//{{V2}}
ORGANIZATION_BLOCK OB1
TITLE= "Cyclic main program"


AUTHOR:nb
FAMILY:nb
NAME:nb
VERSION:1.0


VAR_TEMP
       OB1_EV_CLASS:BYTE //Bits 0-3 = 1 (Coming event), Bits 4-7 = 1 (Event class 1)
       OB1_SCAN_1:BYTE //1 (Cold restart scan 1 of OB 1), 3 (Scan 2-n of OB 1)
       OB1_PRIORITY:BYTE //1 (Priority of 1 is lowest)
       OB1_OB_NUMBR:BYTE //1 (Organization block 1, OB1)
       OB1_RESERVED_1:BYTE //Reserved for system
       OB1_RESERVED_2:BYTE //Reserved for system
       OB1_PREV_CYCLE:INT //Cycle time of previous OB1 scan (milliseconds)
       OB1_MIN_CYCLE:INT //Minimum cycle time of OB1 (milliseconds)
       OB1_MAX_CYCLE:INT //Maximum cycle time of OB1 (milliseconds)
       OB1_DATE_TIME:DATE_AND_TIME //Date and time OB1 started
END_VAR
BEGIN

NETWORK
TITLE=Linja e Start,Stop,Run,Emergjenca dhe dritat e Start && Reset
//{{k}}
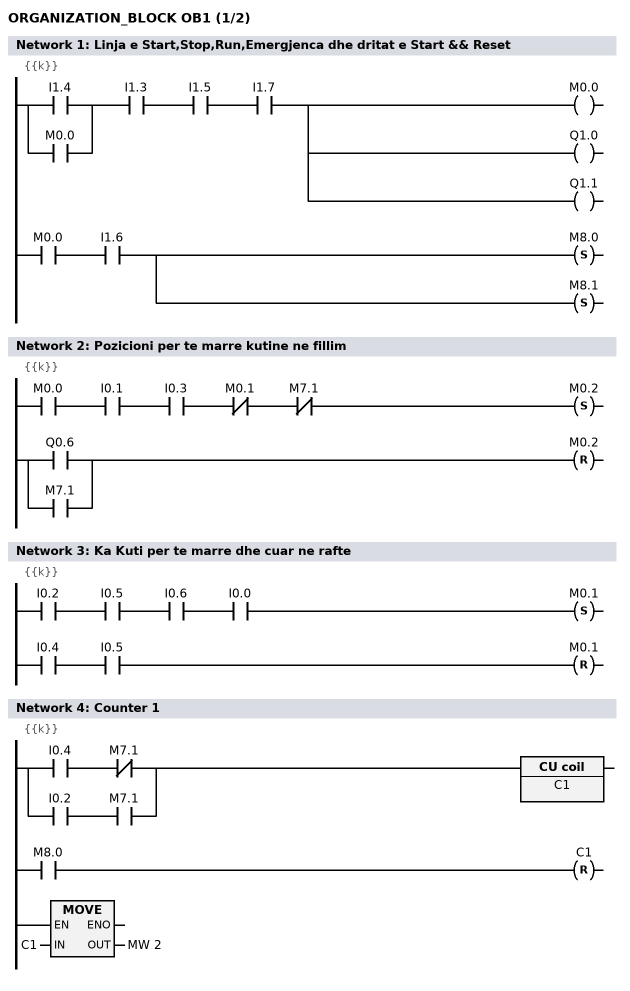

       A(
       O    I1.4
       O    M0.0
       )
       A    I1.3
       A    I1.5
       A    I1.7
       =    M0.0
       =    Q1.0
       =    Q1.1
       A    M0.0
       A    I1.6
       S    M8.0
       S    M8.1
NETWORK
TITLE=Pozicioni per te marre kutine ne fillim
//{{k}}

       A    M0.0
       A    I0.1
       A    I0.3
       AN   M0.1
       AN   M7.1
       S    M0.2
       A(
       O    Q0.6
       O    M7.1
       )
       R    M0.2
NETWORK
TITLE=Ka Kuti per te marre dhe cuar ne rafte
//{{k}}

       A    I0.2
       A    I0.5
       A    I0.6
       A    I0.0
       S    M0.1
       A    I0.4
       A    I0.5
       R    M0.1
NETWORK
TITLE=Counter 1
//{{k}}

       A    I0.4
       AN   M7.1
       O
       A    I0.2
       A    M7.1
       CU   C1
       BLD  101
       NOP  0
       NOP  0
       A    M8.0
       R    C1
       L    C1
       T    MW        2
       NOP  0
       NOP  0
NETWORK
TITLE=Timer per A6 dhe A7
//{{k}}
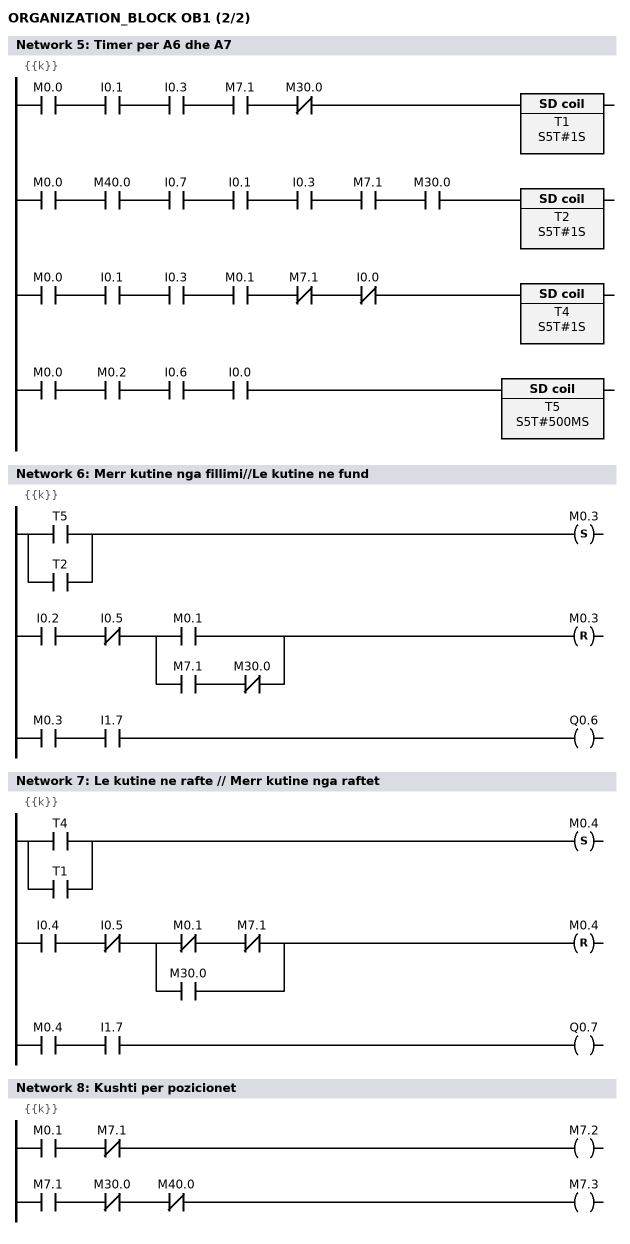

       A    M0.0
       A    I0.1
       A    I0.3
       A    M7.1
       AN   M30.0
       L    S5T#1S
       SD   T1
       A    M0.0
       A    M40.0
       A    I0.7
       A    I0.1
       A    I0.3
       A    M7.1
       A    M30.0
       L    S5T#1S
       SD   T2
       A    M0.0
       A    I0.1
       A    I0.3
       A    M0.1
       AN   M7.1
       AN   I0.0
       L    S5T#1S
       SD   T4
       A    M0.0
       A    M0.2
       A    I0.6
       A    I0.0
       L    S5T#500MS
       SD   T5
NETWORK
TITLE=Merr kutine nga fillimi//Le kutine ne fund
//{{k}}

       O    T5
       O    T2
       S    M0.3
       A    I0.2
       AN   I0.5
       A(
       A    M0.1
       O
       A    M7.1
       AN   M30.0
       )
       R    M0.3
       A    M0.3
       A    I1.7
       =    Q0.6
NETWORK
TITLE=Le kutine ne rafte // Merr kutine nga raftet
//{{k}}

       O    T4
       O    T1
       S    M0.4
       A    I0.4
       AN   I0.5
       A(
       AN   M0.1
       AN   M7.1
       O    M30.0
       )
       R    M0.4
       A    M0.4
       A    I1.7
       =    Q0.7
NETWORK
TITLE=Kushti per pozicionet
//{{k}}

       A    M0.1
       AN   M7.1
       =    M7.2
       A    M7.1
       AN   M30.0
       AN   M40.0
       =    M7.3
NETWORK
TITLE=Pozicioni 1
//{{k}}

       A(
       A    M0.0
       A(
       L    MW        2
       L    0
       ==I
       )
       A    I0.3
       A(
       O    M7.2
       O    M7.3
       )
       S    M0.5
       A    M0.0
       A(
       O    M0.2
       O    M30.0
       )
       )
       R    M0.5
       NOP  0
NETWORK
TITLE=Pozicioni 2
//{{k}}

       A(
       A    M0.0
       A(
       L    MW        2
       L    1
       ==I
       )
       A    I0.3
       A(
       O    M7.2
       O    M7.3
       )
              S    M0.6
       A    M0.0
       A(
       O    M0.2
       O    M30.0
       )
       )
       R    M0.6
       NOP  0
NETWORK
TITLE=Pozicioni 3
//{{k}}

       A(
       A(
       A    M0.0
       A(
       L    MW        2
       L    2
       ==I
       )
       A    I0.3
       A(
       O    M7.2
       O    M7.3
       )

       )
       S    M0.7
       A    M0.0
       A(
       O    M0.2
       O    M30.0
       )
       )
       R    M0.7
       NOP  0
NETWORK
TITLE=Pozicioni 4
//{{k}}

       A(
       A(
       A    M0.0
       A(
       L    MW        2
       L    3
       ==I
       )
       A    I0.3
       A(
       O    M7.2
       O    M7.3
       )
       )
       S    M1.0
       A    M0.0
       A(
       O    M0.2
       O    M30.0
       )
       )
       R    M1.0
       NOP  0
NETWORK
TITLE=Pozicioni 5
//{{k}}

       A(
       A(
       A    M0.0
       A(
       L    MW        2
       L    4
       ==I
       )
       A    I0.3
       A(
       O    M7.2
       O    M7.3
       )

       )
       S    M1.1
       A    M0.0
       A(
       O    M0.2
       O    M30.0
       )
       )
       R    M1.1
       NOP  0
NETWORK
TITLE=Pozicioni 6
//{{k}}

       A(
       A(
       A    M0.0
       A(
       L    MW        2
       L    5
       ==I
       )
       A    I0.3
       A(
       O    M7.2
       O    M7.3
       )

             )
       S    M1.2
       A    M0.0
       A(
       O    M0.2
       O    M30.0
       )
       )
       R    M1.2
       NOP  0
NETWORK
TITLE=Pozicioni 7
//{{k}}

       A(
       A(
       A    M0.0
       A(
       L    MW        2
       L    6
       ==I
       )
       A    I0.3
       A(
       O    M7.2
       O    M7.3
       )


       )
       S    M1.3
       A    M0.0
       A(
       O    M0.2
       O    M30.0
       )
       )
       R    M1.3
       NOP  0
NETWORK
TITLE=Pozicioni 8
//{{k}}

       A(
       A(
       A    M0.0
       A(
       L    MW        2
       L    7
       ==I
       )
       A    I0.3
       A(
       O    M7.2
       O    M7.3
       )


       )
       S    M1.4
       A    M0.0
       A(
       O    M0.2
       O    M30.0
       )
       )
       R    M1.4
       NOP  0
NETWORK
TITLE=Pozicioni 9
//{{k}}

       A(
       A(
       A    M0.0
       A(
       L    MW        2
       L    8
       ==I
       )
       A    I0.3
       A(
       O    M7.2
       O    M7.3
       )


       )
       S    M1.5
       A    M0.0
       A(
       O    M0.2
       O    M30.0
       )
       )
       R    M1.5
       NOP  0
NETWORK
TITLE=Pozicioni 10
//{{k}}

       A(
       A(
       A    M0.0
       A(
       L    MW        2
       L    9
       ==I
       )
       A    I0.3
       A(
       O    M7.2
       O    M7.3
       )

       )
       S    M1.6
       A    M0.0
       A(
       O    M0.2
       O    M30.0
       )
       )
       R    M1.6
       NOP  0
NETWORK
TITLE=Pozicioni 11
//{{k}}

       A(
       A(
       A    M0.0
       A(
       L    MW        2
       L    10
       ==I
       )
       A    I0.3
       A(
       O    M7.2
       O    M7.3
       )


       )
       S    M1.7
       A    M0.0
       A(
       O    M0.2
       O    M30.0
       )
       )
       R    M1.7
       NOP  0
NETWORK
TITLE=Pozicioni 12
//{{k}}

       A(
       A(
       A    M0.0
       A(
       L    MW        2
       L    11
       ==I
       )
       A    I0.3
       A(
       O    M7.2
       O    M7.3
       )

              )
       S    M2.0
       A    M0.0
       A(
       O    M0.2
       O    M30.0
       )
       )
       R    M2.0
       NOP  0
NETWORK
TITLE=Pozicioni 13
//{{k}}

       A(
       A(
       A    M0.0
       A(
       L    MW        2
       L    12
       ==I
       )
       A    I0.3
       A(
       O    M7.2
       O    M7.3
       )


       )
       S    M2.1
       A    M0.0
       A(
       O    M0.2
       O    M30.0
       )
       )
       R    M2.1
       NOP  0
NETWORK
TITLE=Pozicioni 14
//{{k}}

       A(
       A(
       A    M0.0
       A(
       L    MW        2
       L    13
       ==I
       )
       A    I0.3
       A(
       O    M7.2
       O    M7.3
       )

       )
       S    M2.2
       A    M0.0
       A(
       O    M0.2
       O    M30.0
       )
       )
       R    M2.2
       NOP  0
NETWORK
TITLE=Pozicioni 15
//{{k}}

       A(
       A(
       A    M0.0
       A(
       L    MW        2
       L    14
       ==I
       )
       A    I0.3
       A(
       O    M7.2
       O    M7.3
       )

       )
       S    M2.3
       A    M0.0
       A(
       O    M0.2
       O    M30.0
       )
       )
       R    M2.3
       NOP  0
NETWORK
TITLE=Pozicioni 16
//{{k}}

       A(
       A(
       A    M0.0
       A(
       L    MW        2
       L    15
       ==I
       )
       A    I0.3
       A(
       O    M7.2
       O    M7.3
       )


       )
       S    M2.4
       A    M0.0
       A(
       O    M0.2
       O    M30.0
       )
       )
       R    M2.4
       NOP  0
NETWORK
TITLE=Pozicioni 17
//{{k}}

       A(
       A(
       A    M0.0
       A(
       L    MW        2
       L    16
       ==I
       )
       A    I0.3
       A(
       O    M7.2
       O    M7.3
       )


       )
       S    M2.5
       A    M0.0
       A(
       O    M0.2
       O    M30.0
       )
       )
       R    M2.5
       NOP  0
NETWORK
TITLE=Pozicioni 18
//{{k}}

       A(
       A(
       A    M0.0
       A(
       L    MW        2
       L    17
       ==I
       )
       A    I0.3
       A(
       O    M7.2
       O    M7.3
       )


       )
       S    M2.6
       A    M0.0
       A(
       O    M0.2
       O    M30.0
       )
       )
       R    M2.6
       NOP  0
NETWORK
TITLE=Pozicioni 19
//{{k}}

       A(
       A(
       A    M0.0
       A(
       L    MW        2
       L    18
       ==I
       )
       A    I0.3
       A(
       O    M7.2
       O    M7.3
       )


       )
       S    M2.7
       A    M0.0
       A(
       O    M0.2
       O    M30.0
       )
       )
       R    M2.7
       NOP  0
NETWORK
TITLE=Pozicioni 20
//{{k}}

       A(
       A(
       A    M0.0
       A(
       L    MW        2
       L    19
       ==I
       )
       A    I0.3
       A(
       O    M7.2
       O    M7.3
       )


       )
       S    M10.0
       A    M0.0
       A(
       O    M0.2
       O    M30.0
       )
       )
       R    M10.0
       NOP  0
NETWORK
TITLE=Pozicioni 21
//{{k}}

       A(
       A(
       A    M0.0
       A(
       L    MW        2
       L    20
       ==I
       )
       A    I0.3
       A(
       O    M7.2
       O    M7.3
       )

             )
       S    M10.1
       A    M0.0
       A(
       O    M0.2
       O    M30.0
       )
       )
       R    M10.1
       NOP  0
NETWORK
TITLE=Pozicioni 22
//{{k}}

       A(
       A(
       A    M0.0
       A(
       L    MW        2
       L    21
       ==I
       )
       A    I0.3
       A(
       O    M7.2
       O    M7.3
       )


       )
       S    M10.2
       A    M0.0
       A(
       O    M0.2
       O    M30.0
       )
       )
       R    M10.2
       NOP  0
NETWORK
TITLE=Pozicioni 23
//{{k}}

       A(
       A(
       A    M0.0
       A(
       L    MW        2
       L    22
       ==I
       )
       A    I0.3
       A(
       O    M7.2
       O    M7.3
       )


       )
       S    M10.3
       A    M0.0
       A(
       O    M0.2
       O    M30.0
       )
       )
       R    M10.3
       NOP  0
NETWORK
TITLE=Pozicioni 24
//{{k}}

       A(
       A(
       A    M0.0
       A(
       L    MW        2
       L    23
       ==I
       )
       A    I0.3
       A(
       O    M7.2
       O    M7.3
       )


       )
       S    M10.4
       A    M0.0
       A(
       O    M0.2
       O    M30.0
       )
       )
       R    M10.4
       NOP  0
NETWORK
TITLE=Pozicioni 25
//{{k}}

       A(
       A(
       A    M0.0
       A(
       L    MW        2
       L    24
       ==I
       )
       A    I0.3
       A(
       O    M7.2
       O    M7.3
       )


       )
       S    M10.5
       A    M0.0
       A(
       O    M0.2
       O    M30.0
       )
       )
       R    M10.5
       NOP  0
NETWORK
TITLE=Pozicioni 26
//{{k}}

       A(
       A(
       A    M0.0
       A(
       L    MW        2
       L    25
       ==I
       )
       A    I0.3
       A(
       O    M7.2
       O    M7.3
       )


       )
       S    M10.6
       A    M0.0
       A(
       O    M0.2
       O    M30.0
       )
       )
       R    M10.6
       NOP  0
NETWORK
TITLE=Pozicioni 27
//{{k}}

       A(
       A(
       A    M0.0
       A(
       L    MW        2
       L    26
       ==I
       )
       A    I0.3
       A(
       O    M7.2
       O    M7.3
       )

              )
       S    M10.7
       A    M0.0
       A(
       O    M0.2
       O    M30.0
       )
       )
       R    M10.7
       NOP  0
NETWORK
TITLE=Pozicioni 28
//{{k}}

       A(
       A(
       A    M0.0
       A(
       L    MW        2
       L    27
       ==I
       )
       A    I0.3
       A(
       O    M7.2
       O    M7.3
       )


       )
       S    M4.0
       A    M0.0
       A(
       O    M0.2
       O    M30.0
       )
       )
       R    M4.0
       NOP  0
NETWORK
TITLE=Pozicioni 29
//{{k}}

       A(
       A(
       A    M0.0
       A(
       L    MW        2
       L    28
       ==I
       )
       A    I0.3
       A(
       O    M7.2
       O    M7.3
       )


       )
       S    M4.1
       A    M0.0
       A(
       O    M0.2
       O    M30.0
       )
       )
       R    M4.1
       NOP  0
NETWORK
TITLE=Pozicioni 30
//{{k}}

       A(
       A(
       A    M0.0
       A(
       L    MW        2
       L    29
       ==I
       )
       A    I0.3
       A(
       O    M7.2
       O    M7.3
       )


       )
       S    M4.2
       A    M0.0
       A(
       O    M0.2
       O    M30.0
       )
       )
       R    M4.2
       NOP  0
NETWORK
TITLE=Pozicioni 31
//{{k}}

       A(
       A(
       A    M0.0
       A(
       L    MW        2
       L    30
       ==I
       )
       A    I0.3
       A(
       O    M7.2
       O    M7.3
       )

       )
       S    M4.3
       A    M0.0
       A(
       O    M0.2
       O    M30.0
       )
       )
       R    M4.3
       NOP  0
NETWORK
TITLE=Pozicioni 32
//{{k}}

       A(
       A(
       A    M0.0
       A(
       L    MW        2
       L    31
       ==I
       )
       A    I0.3
       A(
       O    M7.2
       O    M7.3
       )

       )
       S    M4.4
       A    M0.0
       A(
       O    M0.2
       O    M30.0
       )
       )
       R    M4.4
       NOP  0
NETWORK
TITLE=Pozicioni 33
//{{k}}

       A(
       A(
       A    M0.0
       A(
       L    MW        2
       L    32
       ==I
       )
       A    I0.3
       A(
       O    M7.2
       O    M7.3
       )

       )
       S    M4.5
       A    M0.0
       A(
       O    M0.2
       O    M30.0
       )
       )
       R    M4.5
       NOP  0
NETWORK
TITLE=Pozicioni 34
//{{k}}

       A(
       A(
       A    M0.0
       A(
       L    MW        2
       L    33
       ==I
       )
       A    I0.3
       A(
       O    M7.2
       O    M7.3
       )

       )
       S    M4.6
       A    M0.0
       A(
       O    M0.2
       O    M30.0
       )
       )
       R    M4.6
       NOP  0
NETWORK
TITLE=Pozicioni 35
//{{k}}

       A(
       A(
       A    M0.0
       A(
       L    MW        2
       L    34
       ==I
       )
       A    I0.3
       A(
       O    M7.2
       O    M7.3
       )

       )
       S    M4.7
       A    M0.0
       A(
       O    M0.2
       O    M30.0
       )
       )
       R    M4.7
       NOP  0
NETWORK
TITLE=Pozicioni 36
//{{k}}

       A(
       A(
       A    M0.0
       A(
       L    MW        2
       L    35
       ==I
       )
       A    I0.3
       A(
       O    M7.2
       O    M7.3
       )


       )
       S    M5.0
       A    M0.0
       A(
       O    M0.2
       O    M30.0
       )
       )
       R    M5.0
       NOP  0
NETWORK
TITLE=Pozicioni 37
//{{k}}

       A(
       A(
       A    M0.0
       A(
       L    MW        2
       L    36
       ==I
       )
       A    I0.3
       A(
       O    M7.2
       O    M7.3
       )


       )
       S    M5.1
       A    M0.0
       A(
       O    M0.2
       O    M30.0
       )
       )
       R    M5.1
       NOP  0
NETWORK
TITLE=Pozicioni 38
//{{k}}

       A(
       A(
       A    M0.0
       A(
       L    MW        2
       L    37
       ==I
       )
       A    I0.3
       A(
       O    M7.2
       O    M7.3
       )


       )
       S    M5.2
       A    M0.0
       A(
       O    M0.2
       O    M30.0
       )
       )
       R    M5.2
       NOP  0
NETWORK
TITLE=Pozicioni 39
//{{k}}

       A(
       A(
       A    M0.0
       A(
       L    MW        2
       L    38
       ==I
       )

       A    I0.3
       A(
       O    M7.2
       O    M7.3
       )

       )

       S    M5.3
       A    M0.0
       A(
       O    M0.2
       O    M30.0
       )
       )
       R    M5.3
       NOP  0
NETWORK
TITLE=Pozicioni 40
//{{k}}

       A(
       A(
       A    M0.0
       A(
       L    MW        2
       L    39
       ==I
       )
       A    I0.3
       A(
       O    M7.2
       O    M7.3
       )

             )
       S    M5.4
       A    M0.0
       A(
       O    M0.2
       O    M30.0
       )
       )
       R    M5.4
       NOP  0
NETWORK
TITLE=Pozicioni 41
//{{k}}

       A(
       A(
       A    M0.0
       A(
       L    MW        2
       L    40
       ==I
       )
       A    I0.3
       A(
       O    M7.2
       O    M7.3
       )

       )
       S    M5.5
       A    M0.0
       A(
       O    M0.2
       O    M30.0
       )
       )
       R    M5.5
       NOP  0
NETWORK
TITLE=Pozicioni 42
//{{k}}

       A(
       A(
       A    M0.0
       A(
       L    MW        2
       L    41
       ==I
       )
       A    I0.3
       A(
       O    M7.2
       O    M7.3
       )

             )
       S    M5.6
       A    M0.0
       A(
       O    M0.2
       O    M30.0
       )
       )
       R    M5.6
       NOP  0
NETWORK
TITLE=Pozicioni 43
//{{k}}

       A(
       A(
       A    M0.0
       A(
       L    MW        2
       L    42
       ==I
       )
       A    I0.3
       A(
       O    M7.2
       O    M7.3
       )

              )
       S    M5.7
       A    M0.0
       A(
       O    M0.2
       O    M30.0
       )
       )
       R    M5.7
       NOP  0
NETWORK
TITLE=Pozicioni 44
//{{k}}

       A(
       A(
       A    M0.0
       A(
       L    MW        2
       L    43
       ==I
       )
       A    I0.3
       A(
       O    M7.2
       O    M7.3
       )

              )
       S    M6.0
       A    M0.0
       A(
       O    M0.2
       O    M30.0
       )
       )
       R    M6.0
       NOP  0
NETWORK
TITLE=Pozicioni 45
//{{k}}

       A(
       A(
       A    M0.0
       A(
       L    MW        2
       L    44
       ==I
       )
       A    I0.3
       A(
       O    M7.2
       O    M7.3
       )


       )
       S    M6.1
       A    M0.0
       A(
       O    M0.2
       O    M30.0
       )
       )
       R    M6.1
       NOP  0
NETWORK
TITLE=Pozicioni 46
//{{k}}

       A(
       A(
       A    M0.0
       A(
       L    MW        2
       L    45
       ==I
       )
       A    I0.3
       A(
       O    M7.2
       O    M7.3
       )

              )
       S    M6.2
       A    M0.0
       A(
       O    M0.2
       O    M30.0
       )
       )
       R    M6.2
       NOP  0
NETWORK
TITLE=Pozicioni 47
//{{k}}

       A(
       A(
       A    M0.0
       A(
       L    MW        2
       L    46
       ==I
       )
       A    I0.3
       A(
       O    M7.2
       O    M7.3
       )

              )
       S    M6.3
       A    M0.0
       A(
       O    M0.2
       O    M30.0
       )
       )
       R    M6.3
       NOP  0
NETWORK
TITLE=Pozicioni 48
//{{k}}

       A(
       A(
       A    M0.0
       A(
       L    MW        2
       L    47
       ==I
       )
       A    I0.3
       A(
       O    M7.2
       O    M7.3
       )


       )
       S    M6.4
       A    M0.0
       A(
       O    M0.2
       O    M30.0
       )
       )
       R    M6.4
       NOP  0
NETWORK
TITLE=Pozicioni 49
//{{k}}

       A(
       A(
       A    M0.0
       A(
       L    MW        2
       L    48
       ==I
       )
       A    I0.3
       A(
       O    M7.2
       O    M7.3
       )


       )
       S    M6.5
       A    M0.0
       A(
       O    M0.2
       O    M30.0
       )
       )
       R    M6.5
       NOP  0
NETWORK
TITLE=Pozicioni 50
//{{k}}

       A(
       A(
       A    M0.0
       A(
       L    MW        2
       L    49
       ==I
       )
       A    I0.3
       A(
       O    M7.2
       O    M7.3
       )

             )
       S    M6.6
       A    M0.0
       A(
       O    M0.2
       O    M30.0
       )
       )
       R    M6.6
       NOP  0
NETWORK
TITLE=Actuator 0
//{{k}}
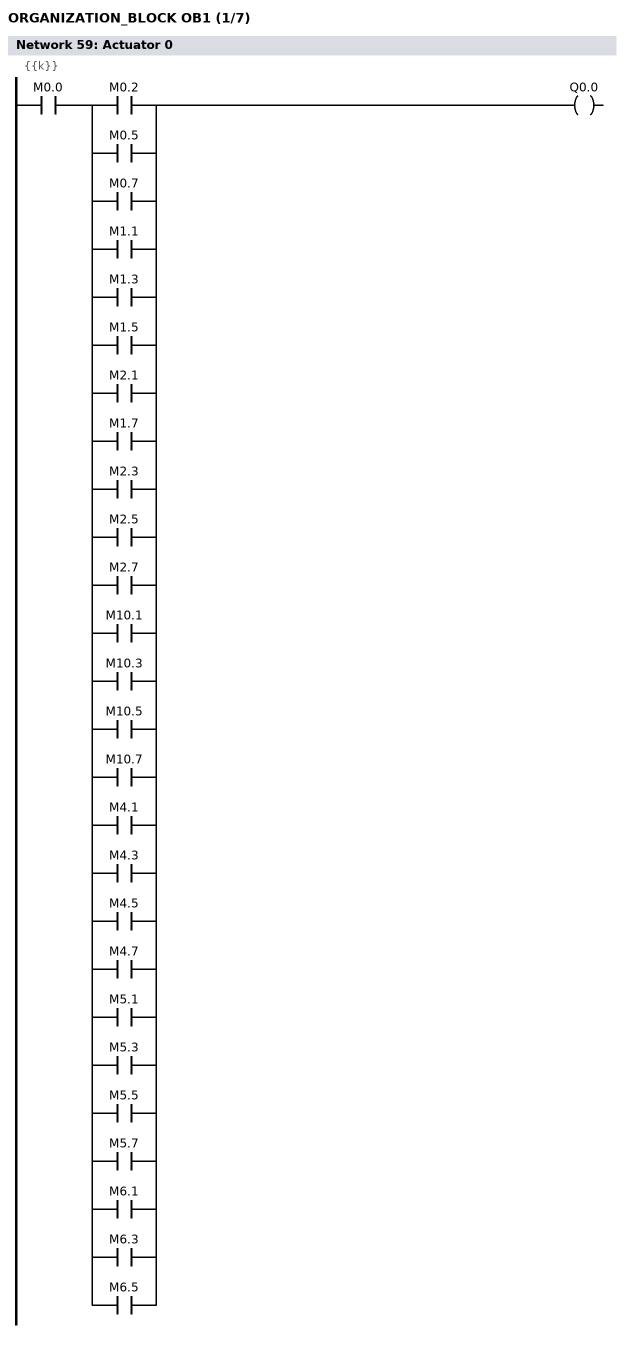

       A    M0.0
       A(
       O    M0.2
       O    M0.5
       O    M0.7
       O    M1.1
       O    M1.3
       O    M1.5
       O    M2.1
       O    M1.7
       O    M2.3
       O    M2.5
       O    M2.7
       O    M10.1
       O    M10.3
       O    M10.5
       O    M10.7
       O    M4.1
       O    M4.3
       O    M4.5
       O    M4.7
       O    M5.1
       O    M5.3
       O    M5.5
       O    M5.7
       O    M6.1
       O    M6.3
       O    M6.5
       )
       =    Q0.0
NETWORK
TITLE=Actuator 1
//{{k}}
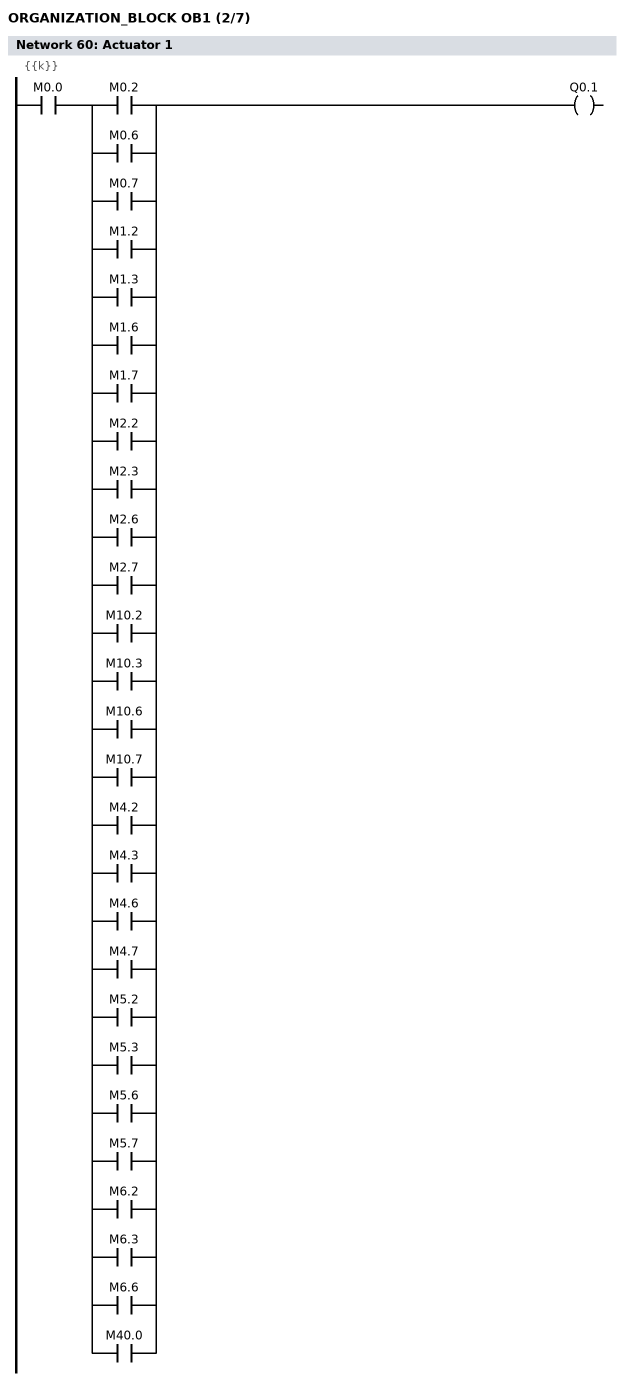

       A    M0.0
       A(
       O    M0.2
       O    M0.6
       O    M0.7
       O    M1.2
       O    M1.3
       O    M1.6
       O    M1.7
       O    M2.2
       O    M2.3
       O    M2.6
       O    M2.7
       O    M10.2
       O    M10.3
       O    M10.6
       O    M10.7
       O    M4.2
       O    M4.3
       O    M4.6
       O    M4.7
       O    M5.2
       O    M5.3
       O    M5.6
       O    M5.7
       O    M6.2
       O    M6.3
       O    M6.6
       O    M40.0
       )
       =    Q0.1
NETWORK
TITLE=Actuator 2
//{{k}}
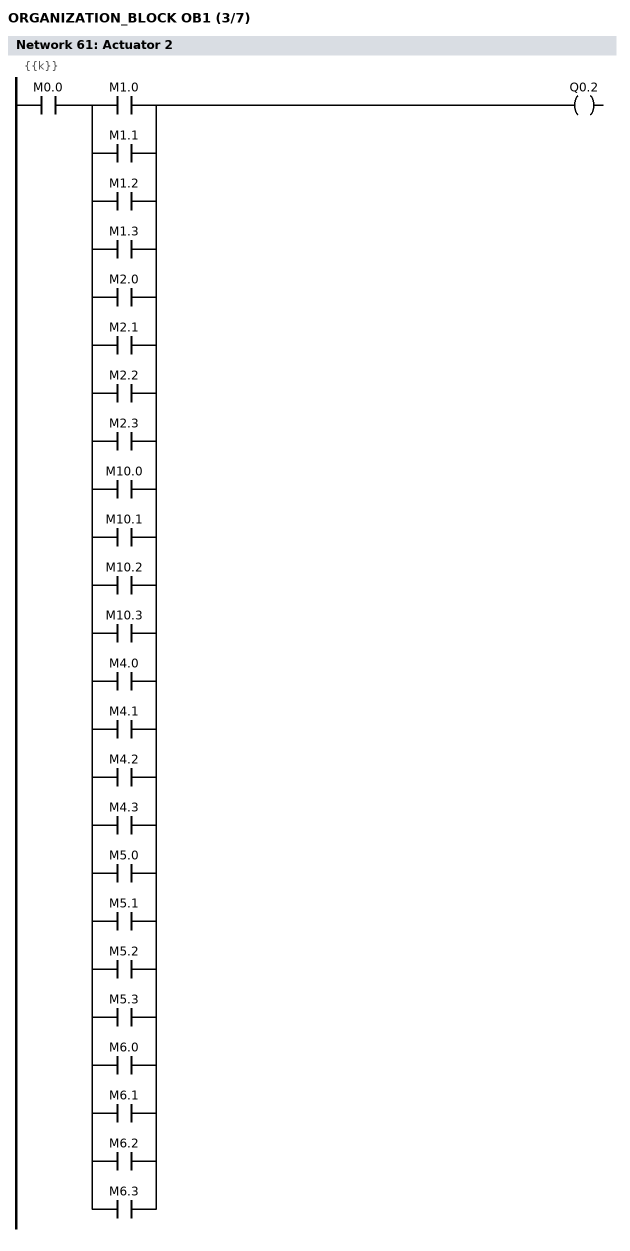

       A    M0.0
       A(
       O    M1.0
       O    M1.1
       O    M1.2
       O    M1.3
       O    M2.0
       O    M2.1
       O    M2.2
       O    M2.3
       O    M10.0
       O    M10.1
       O    M10.2
       O    M10.3
       O    M4.0
       O    M4.1
       O    M4.2
       O    M4.3
       O    M5.0
       O    M5.1
       O    M5.2
       O    M5.3
       O    M6.0
       O    M6.1
       O    M6.2
       O    M6.3
       )
       =    Q0.2
NETWORK
TITLE=Actuator 3
//{{k}}
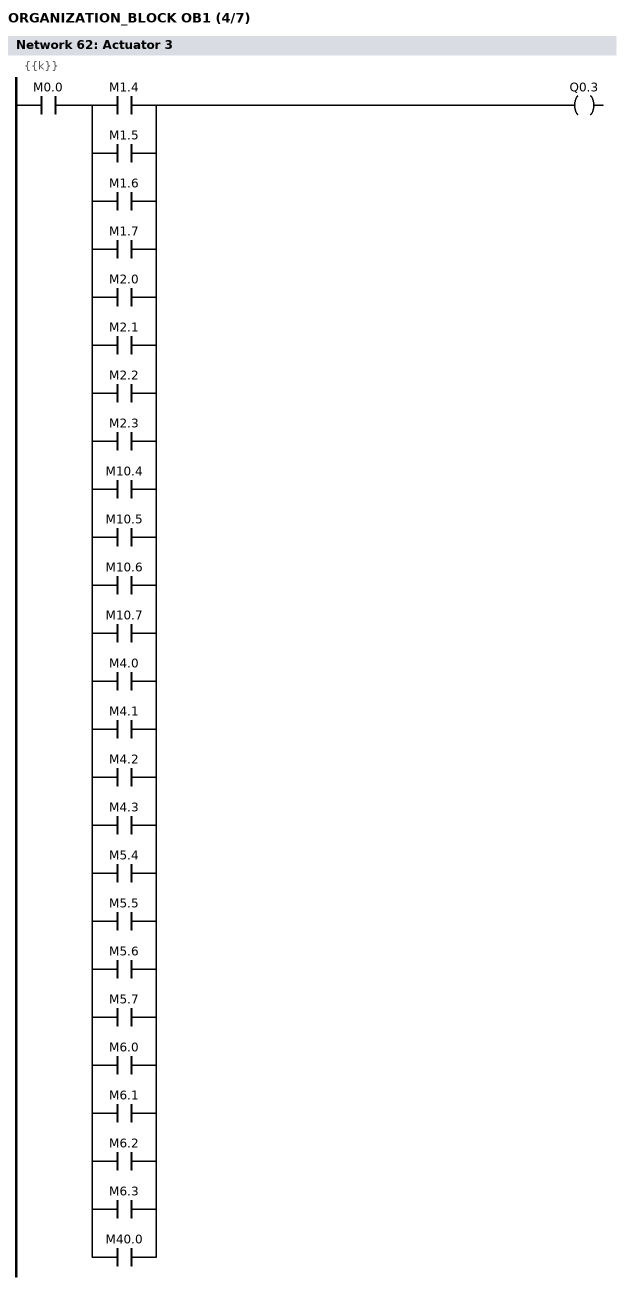

       A    M0.0
       A(
       O    M1.4
       O    M1.5
       O    M1.6
       O    M1.7
       O    M2.0
       O    M2.1
       O    M2.2
       O    M2.3
       O    M10.4
       O    M10.5
       O    M10.6
       O    M10.7
       O    M4.0
       O    M4.1
       O    M4.2
       O    M4.3
       O    M5.4
       O    M5.5
       O    M5.6
       O    M5.7
       O    M6.0
       O    M6.1
       O    M6.2
       O    M6.3
       O    M40.0
       )
       =    Q0.3
NETWORK
TITLE=Actuator 4
//{{k}}
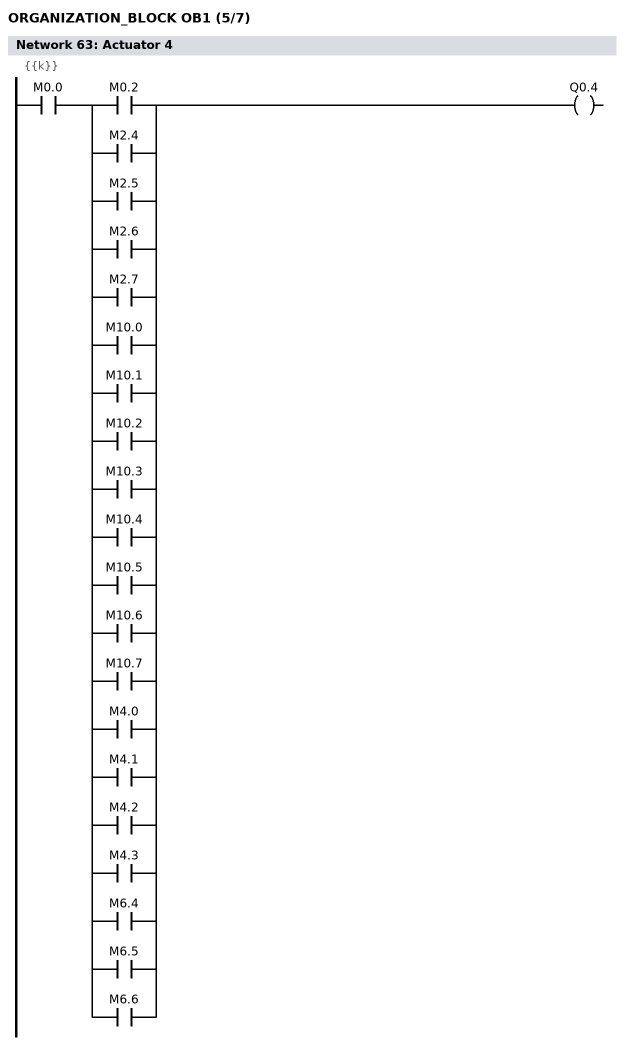

       A    M0.0
       A(
       O    M0.2
       O    M2.4
       O    M2.5
       O    M2.6
       O    M2.7
       O    M10.0
       O    M10.1
       O    M10.2
       O    M10.3
       O    M10.4
       O    M10.5
       O    M10.6
       O    M10.7
       O    M4.0
       O    M4.1
       O    M4.2
       O    M4.3
       O    M6.4
       O    M6.5
       O    M6.6
       )
       =    Q0.4
NETWORK
TITLE=Actuator 5
//{{k}}
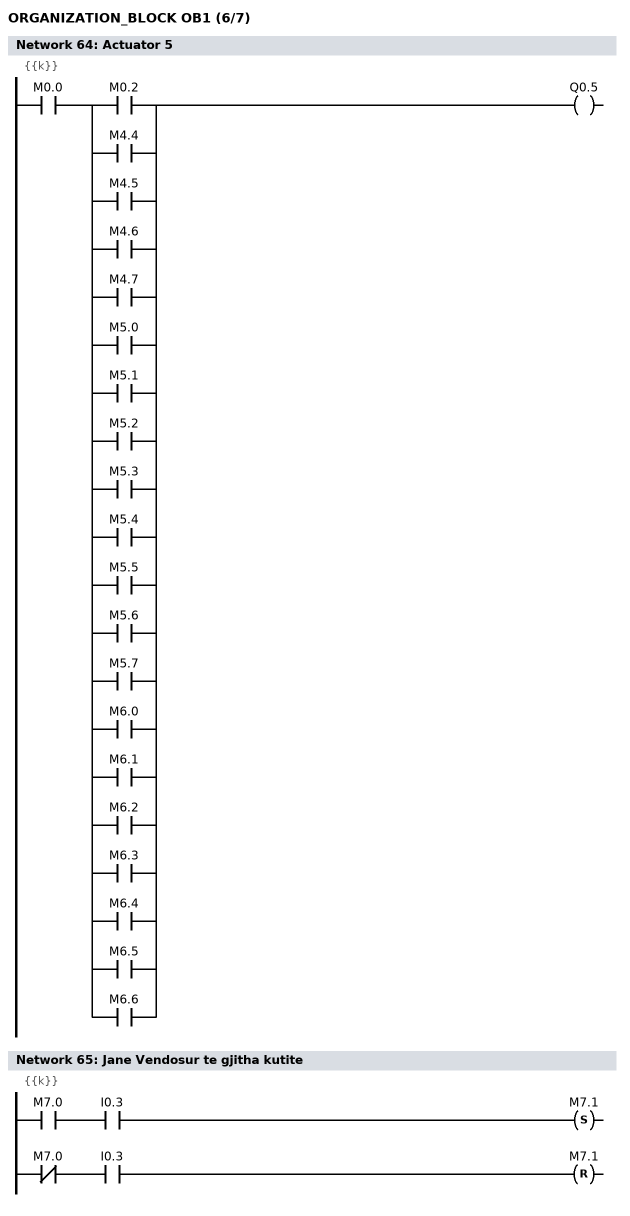

       A    M0.0
       A(
       O    M0.2
       O    M4.4
       O    M4.5
       O    M4.6
       O    M4.7
       O    M5.0
       O    M5.1
       O    M5.2
       O    M5.3
       O    M5.4
       O    M5.5
       O    M5.6
       O    M5.7
       O    M6.0
       O    M6.1
       O    M6.2
       O    M6.3
       O    M6.4
       O    M6.5
       O    M6.6
       )
       =    Q0.5
NETWORK
TITLE=Jane Vendosur te gjitha kutite
//{{k}}

       A    M7.0
       A    I0.3
       S    M7.1
       AN   M7.0
       A    I0.3
       R    M7.1
NETWORK
TITLE=Merret Kutia nga rafti
//{{k}}
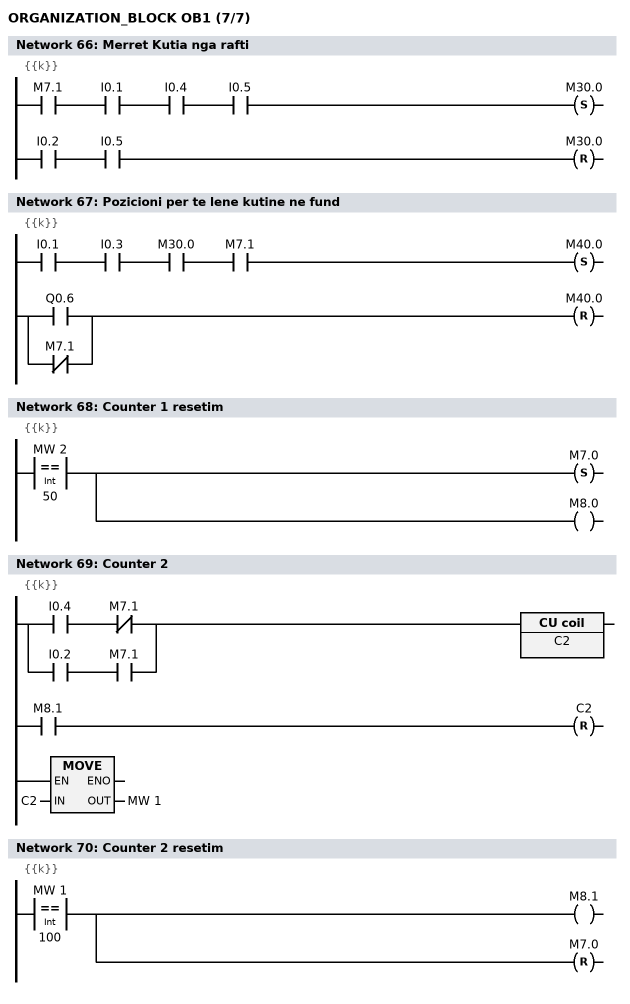

       A    M7.1
       A    I0.1
       A    I0.4
       A    I0.5
       S    M30.0
       A    I0.2
       A    I0.5
       R    M30.0
NETWORK
TITLE=Pozicioni per te lene kutine ne fund
//{{k}}

       A    I0.1
       A    I0.3
       A    M30.0
       A    M7.1
       S    M40.0
       A(
       O    Q0.6
       ON   M7.1
       )
       R    M40.0
NETWORK
TITLE=Counter 1 resetim
//{{k}}

       A(
       L    MW        2
       L    50
       ==I
       )
       S    M7.0
       =    M8.0
NETWORK
TITLE=Counter 2
//{{k}}

       A    I0.4
       AN   M7.1
       O
       A    I0.2
       A    M7.1
       CU   C2
       BLD  101
       NOP  0
       NOP  0
       A    M8.1
       R    C2
       L    C2
       T    MW        1
       NOP  0
       NOP  0
NETWORK
TITLE= Counter 2 resetim
//{{k}}

       A(
       L    MW        1
       L    100
       ==I
       )
       =    M8.1
       R    M7.0
END_ORGANIZATION_BLOCK
